// TIA Portal V21 export
DATA_BLOCK "Percorso"   // DB9
{ S7_Optimized_Access := 'TRUE' }
// stored: MemoryReserve 100
   VAR RETAIN
      Stazione { S7_SetPoint := 'True'} : Array[0.."K_NumStazione"] of "Std_Stazione";
   END_VAR
   VAR
      Hmi : Struct
         Visibilità : Struct
            PompaAcidificazioneVascaEvaporati : Struct
               VascaEvaporati : Bool := FALSE;
            END_STRUCT;
            Acidificazione1 : Struct
               Serpentino : Bool := FALSE;
               VascaPolpa1 : Bool := FALSE;
               VascaPolpa2 : Bool := FALSE;
            END_STRUCT;
            Acidificazione2 : Struct
               Serpentino : Bool := FALSE;
               VascaPolpa1 : Bool := FALSE;
               VascaPolpa2 : Bool := FALSE;
            END_STRUCT;
            Acidificazione3 : Struct
               Serpentino : Bool := FALSE;
               VascaPolpa1 : Bool := FALSE;
               VascaPolpa2 : Bool := FALSE;
               VascaMix : Bool := FALSE;
            END_STRUCT;
            Acidificazione4 : Struct
               Serpentino : Bool := FALSE;
               VascaPolpa1 : Bool := FALSE;
               VascaPolpa2 : Bool := FALSE;
            END_STRUCT;
            BermaProntoFresco : Struct
               CatelliLogicon : Bool := FALSE;
               CFT10t : Bool := FALSE;
               CatelliOhmico : Bool := FALSE;
               Goglio : Bool := FALSE;
            END_STRUCT;
            BermaPomodoro : Struct
               CatelliLogicon : Bool := FALSE;
               CFT10t : Bool := FALSE;
               CatelliOhmico : Bool := FALSE;
               Goglio : Bool := FALSE;
            END_STRUCT;
            Cernita1 : Struct
               IFT6 : Bool := FALSE;
               TrituratoD1 : Bool := FALSE;
            END_STRUCT;
            CFT_MVRAEstrazione1 : Struct
               VascaDecanter : Bool := FALSE;
               Vasca30Quintali : Bool := FALSE;
               VascaEvaporati : Bool := FALSE;
               CFT10t : Bool := FALSE;
               CatelliConcentrato : Bool := FALSE;
               CatelliOhmico : Bool := FALSE;
               BermaPomodoro : Bool := FALSE;
               BermaProntoFresco : Bool := FALSE;
               Ghizzoni : Bool := FALSE;
               PastorizzatoreGoglio2 : Bool := FALSE;
            END_STRUCT;
            CFT_MVRAEstrazione2 : Struct
               VascaDecanter : Bool := FALSE;
               Vasca30Quintali : Bool := FALSE;
               VascaEvaporati : Bool := FALSE;
               VascaSemiconcentrato : Bool := FALSE;
               CFT10t : Bool := FALSE;
               CatelliLogicon : Bool := FALSE;
               CatelliConcentrato : Bool := FALSE;
               CatelliOhmico : Bool := FALSE;
               Goglio : Bool := FALSE;
               BermaPomodoro : Bool := FALSE;
               BermaProntoFresco : Bool := FALSE;
               Ghizzoni : Bool := FALSE;
               PastorizzatoreGoglio2 : Bool := FALSE;
            END_STRUCT;
            CFT_MVRBEstrazione1 : Struct
               VascaDecanter : Bool := FALSE;
               Vasca30Quintali : Bool := FALSE;
               VascaPolpa1 : Bool := FALSE;
               VascaSemiconcentrato : Bool := FALSE;
               CFT10t : Bool := FALSE;
               CatelliLogicon : Bool := FALSE;
               CatelliOhmico : Bool := FALSE;
               Goglio : Bool := FALSE;
               BermaPomodoro : Bool := FALSE;
               BermaProntoFresco : Bool := FALSE;
               Ghizzoni : Bool := FALSE;
               PastorizzatoreGoglio2 : Bool := FALSE;
            END_STRUCT;
            CFT_MVRBFinitore1 : Struct
               VascaDecanter : Bool := FALSE;
               Vasca30Quintali : Bool := FALSE;
               VascaPolpa1 : Bool := FALSE;
               VascaSemiconcentrato : Bool := FALSE;
               CFT10t : Bool := FALSE;
               CatelliLogicon : Bool := FALSE;
               CatelliConcentrato : Bool := FALSE;
               CatelliOhmico : Bool := FALSE;
               Goglio : Bool := FALSE;
               BermaPomodoro : Bool := FALSE;
               BermaProntoFresco : Bool := FALSE;
               Ghizzoni : Bool := FALSE;
               PastorizzatoreGoglio2 : Bool := FALSE;
            END_STRUCT;
            CFT_MVRBFinitore2 : Struct
               VascaEvaporati : Bool := FALSE;
               CatelliConcentrato : Bool := FALSE;
               FBR200Kg : Bool := FALSE;
            END_STRUCT;
            CocleaIFT1_2 : Struct
               IFT1 : Bool := FALSE;
               IFT2 : Bool := FALSE;
            END_STRUCT;
            D1 : Struct
               PompaAlimentazioneHB1 : Bool := FALSE;
               PompaAlimentazioneHB2 : Bool := FALSE;
               PompaAlimentazioneHB1_HB2 : Bool := FALSE;
            END_STRUCT;
            D2 : Struct
               PompaAlimentazioneHB1 : Bool := FALSE;
               PompaAlimentazioneHB2 : Bool := FALSE;
               PompaAlimentazioneHB1_HB2 : Bool := FALSE;
            END_STRUCT;
            VascaDecanter1 : Struct
               VascaCrema : Bool := FALSE;
            END_STRUCT;
            VascaDecanter2 : Struct
               VascaCrema : Bool := FALSE;
            END_STRUCT;
            VascaDecanter3 : Struct
               VascaCrema : Bool := FALSE;
            END_STRUCT;
            Ghizzoni : Struct
               CFT10t : Bool := FALSE;
               CatelliLogicon : Bool := FALSE;
               CatelliOhmico : Bool := FALSE;
               Goglio : Bool := FALSE;
            END_STRUCT;
            IFT3 : Struct
               Lince1 : Bool := FALSE;
               Lince2 : Bool := FALSE;
               Lince3 : Bool := FALSE;
            END_STRUCT;
            IFT5 : Struct
               Lince1 : Bool := FALSE;
               Lince3 : Bool := FALSE;
            END_STRUCT;
            IFT6 : Struct
               Lince1 : Bool := FALSE;
               Lince2 : Bool := FALSE;
               Lince3 : Bool := FALSE;
            END_STRUCT;
            Lince1 : Struct
               Serpentino : Bool := FALSE;
               VascaPolpa1 : Bool := FALSE;
               VascaPolpa2 : Bool := FALSE;
            END_STRUCT;
            Lince2 : Struct
               Serpentino : Bool := FALSE;
               VascaPolpa1 : Bool := FALSE;
               VascaPolpa2 : Bool := FALSE;
            END_STRUCT;
            Lince3 : Struct
               Serpentino : Bool := FALSE;
               VascaPolpa1 : Bool := FALSE;
               VascaPolpa2 : Bool := FALSE;
               VascaMIx : Bool := FALSE;
            END_STRUCT;
            Lince4 : Struct
               Serpentino : Bool := FALSE;
               VascaPolpa1 : Bool := FALSE;
               VascaPolpa2 : Bool := FALSE;
            END_STRUCT;
            PICO1 : Struct
               CFT10t : Bool := FALSE;
               CatelliLogicon : Bool := FALSE;
               CatelliOhmico : Bool := FALSE;
               Goglio : Bool := FALSE;
               BermaPomodoro : Bool := FALSE;
               BermaProntoFresco : Bool := FALSE;
               Ghizzoni : Bool := FALSE;
               FBR200Kg : Bool := FALSE;
               PastorizzatoreGoglio2 : Bool := FALSE;
            END_STRUCT;
            PICO2 : Struct
               CFT10t : Bool := FALSE;
               CatelliLogicon : Bool := FALSE;
               CatelliConcentrato : Bool := FALSE;
               CatelliOhmico : Bool := FALSE;
               Goglio : Bool := FALSE;
               BermaPomodoro : Bool := FALSE;
               BermaProntoFresco : Bool := FALSE;
               Ghizzoni : Bool := FALSE;
               FBR200Kg : Bool := FALSE;
               PastorizzatoreGoglio2 : Bool := FALSE;
            END_STRUCT;
            PompaAlimentazioneDecanter : Struct
               VascaDecanter : Bool := FALSE;
            END_STRUCT;
            PompaAlimentazioneHB1 : Struct
               HB1 : Bool := FALSE;
               HB2 : Bool := FALSE;
            END_STRUCT;
            PompaAlimentazioneHB2 : Struct
               HB1 : Bool := FALSE;
               HB2 : Bool := FALSE;
               HB3 : Bool := FALSE;
            END_STRUCT;
            PompaAlimentazioneHB1_HB2 : Struct
               HB1 : Bool := FALSE;
               HB2 : Bool := FALSE;
            END_STRUCT;
            PompaAlimentazioneHB3 : Struct
               HB3 : Bool := FALSE;
            END_STRUCT;
            PompaInvio1 : Struct
               VascaMix : Bool := FALSE;
               CatelliConcentrato : Bool := FALSE;
               CatelliOhmico : Bool := FALSE;
               BermaPomodoro : Bool := FALSE;
               Ghizzoni : Bool := FALSE;
            END_STRUCT;
            PompaInvio2 : Struct
               CFT10t : Bool := FALSE;
               CatelliLogicon : Bool := FALSE;
               CatelliOhmico : Bool := FALSE;
               PastorizzatoreGoglio2 : Bool := FALSE;
               Ghizzoni : Bool := FALSE;
            END_STRUCT;
            PompaInvio3 : Struct
               FMCPolpa : Bool := FALSE;
               BermaPomodoro : Bool := FALSE;
            END_STRUCT;
            PompaInvio4 : Struct
               FMCPolpa : Bool := FALSE;
            END_STRUCT;
            PompaInvio5 : Struct
               CFT10t : Bool := FALSE;
               CatelliLogicon : Bool := FALSE;
               CatelliOhmico : Bool := FALSE;
               BermaPomodoro : Bool := FALSE;
               BermaProntoFresco : Bool := FALSE;
               Ghizzoni : Bool := FALSE;
               Goglio : Bool := FALSE;
            END_STRUCT;
            PompaInvio6 : Struct
               BermaProntoFresco : Bool := FALSE;
               Ghizzoni : Bool := FALSE;
               Goglio : Bool := FALSE;
               FBR200Kg : Bool := FALSE;
               PastorizzatoreGoglio2 : Bool := FALSE;
            END_STRUCT;
            PompaInvio7 : Struct
               CatelliLogicon : Bool := FALSE;
               CatelliOhmico : Bool := FALSE;
               Goglio : Bool := FALSE;
               BermaProntoFresco : Bool := FALSE;
               Ghizzoni : Bool := FALSE;
               FBR200Kg : Bool := FALSE;
               PastorizzatoreGoglio2 : Bool := FALSE;
            END_STRUCT;
            PompaNastroIFT1_2 : Struct
               D1 : Bool := FALSE;
               D2 : Bool := FALSE;
            END_STRUCT;
            PompaRecuperoIFT1 : Struct
               SgrondatoreP54 : Bool := FALSE;
               SgrondatoreP55 : Bool := FALSE;
            END_STRUCT;
            PompaRecuperoIFT2 : Struct
               SgrondatoreP54 : Bool := FALSE;
               SgrondatoreP55 : Bool := FALSE;
            END_STRUCT;
            PompaRecuperoPizza : Struct
               VascaDecanter : Bool := FALSE;
            END_STRUCT;
            Salsina1 : Struct
               Serpentino : Bool := FALSE;
               VascaPolpa1 : Bool := FALSE;
               VascaPolpa2 : Bool := FALSE;
            END_STRUCT;
            Salsina2 : Struct
               Serpentino : Bool := FALSE;
               VascaPolpa1 : Bool := FALSE;
               VascaPolpa2 : Bool := FALSE;
            END_STRUCT;
            Salsina3 : Struct
               Serpentino : Bool := FALSE;
               VascaPolpa1 : Bool := FALSE;
               VascaPolpa2 : Bool := FALSE;
               VascaMIx : Bool := FALSE;
            END_STRUCT;
            Salsina4 : Struct
               Serpentino : Bool := FALSE;
               VascaPolpa1 : Bool := FALSE;
               VascaPolpa2 : Bool := FALSE;
            END_STRUCT;
            Scrambler : Struct
               Lince1 : Bool := FALSE;
               Lince2 : Bool := FALSE;
               Lince3 : Bool := FALSE;
            END_STRUCT;
            Separapelli1Sx : Struct
               IFT3 : Bool := FALSE;
               IFT4 : Bool := FALSE;
               IFT5 : Bool := FALSE;
               Scrambler : Bool := FALSE;
            END_STRUCT;
            Separapelli2Dx : Struct
               IFT3 : Bool := FALSE;
               IFT4 : Bool := FALSE;
               IFT5 : Bool := FALSE;
               Scrambler : Bool := FALSE;
            END_STRUCT;
            Serpentino : Struct
               PompaInvio1 : Bool := FALSE;
               PompaInvio2 : Bool := FALSE;
               PompaInvio3 : Bool := FALSE;
               PompaInvio4 : Bool := FALSE;
               PompaInvio5 : Bool := FALSE;
            END_STRUCT;
            SgrondatoreP54 : Struct
               Lince1 : Bool := FALSE;
               Lince2 : Bool := FALSE;
               Lince3 : Bool := FALSE;
            END_STRUCT;
            SgrondatoreP55 : Struct
               Lince2 : Bool := FALSE;
               Lince3 : Bool := FALSE;
            END_STRUCT;
            "T150_1/2EffettoP05" : Struct
               VascaDecanter : Bool := FALSE;
               VascaEvaporati : Bool := FALSE;
               VascaPolpa1 : Bool := FALSE;
               Ghizzoni : Bool := FALSE;
               VascaSemiconcentrato : Bool := FALSE;
            END_STRUCT;
            "T150_1/2EffettoP07" : Struct
               VascaDecanter : Bool := FALSE;
               VascaEvaporati : Bool := FALSE;
               VascaPolpa1 : Bool := FALSE;
               CatelliOhmico : Bool := FALSE;
               Ghizzoni : Bool := FALSE;
               VascaSemiconcentrato : Bool := FALSE;
               BermaPomodoro : Bool := FALSE;
               BermaProntoFresco : Bool := FALSE;
            END_STRUCT;
            T150_3EffettofinitoreP02 : Struct
               VascaEvaporati : Bool := FALSE;
               VascaPolpa1 : Bool := FALSE;
               CatelliConcentrato : Bool := FALSE;
               CatelliOhmico : Bool := FALSE;
               VascaSemiconcentrato : Bool := FALSE;
               BermaPomodoro : Bool := FALSE;
               VascaDecanter : Bool := FALSE;
            END_STRUCT;
            TorchioSgrondatoreP54 : Struct
               Lince3 : Bool := FALSE;
            END_STRUCT;
            TorchioScrambler : Struct
               Lince1 : Bool := FALSE;
            END_STRUCT;
            TrituratoD1 : Struct
               D1 : Bool := FALSE;
            END_STRUCT;
            TrituratoD2 : Struct
               D2 : Bool := FALSE;
            END_STRUCT;
            TrituratoBrovatrice : Struct
               D1 : Bool := FALSE;
               D2 : Bool := FALSE;
            END_STRUCT;
            Vasca30Quintali : Struct
               Serpentino : Bool := FALSE;
            END_STRUCT;
            VascaDecanter : Struct
               VascaEvaporati : Bool := FALSE;
               Vasca30Quintali : Bool := FALSE;
               VascaPolpa1 : Bool := FALSE;
               Decanter1 : Bool := FALSE;
               Decanter2 : Bool := FALSE;
               Decanter3 : Bool := FALSE;
            END_STRUCT;
            VascaEvaporatiP134 : Struct
               CatelliOhmico : Bool := FALSE;
            END_STRUCT;
            VascaEvaporatiP135 : Struct
               CatelliConcentrato : Bool := FALSE;
            END_STRUCT;
            VascaMix : Struct
               PICO1 : Bool := FALSE;
               PICO2 : Bool := FALSE;
            END_STRUCT;
            VascaPolpa1 : Struct
               PompaInvio1 : Bool := FALSE;
               PompaInvio2 : Bool := FALSE;
               PompaInvio3 : Bool := FALSE;
               PompaInvio4 : Bool := FALSE;
               PompaInvio5 : Bool := FALSE;
               PompaInvio6 : Bool := FALSE;
               PompaInvio7 : Bool := FALSE;
            END_STRUCT;
            VascaPolpa2 : Struct
               PompaInvio1 : Bool := FALSE;
               PompaInvio2 : Bool := FALSE;
               PompaInvio3 : Bool := FALSE;
               PompaInvio4 : Bool := FALSE;
               PompaInvio5 : Bool := FALSE;
               PompaInvio6 : Bool := FALSE;
               PompaInvio7 : Bool := FALSE;
            END_STRUCT;
            PompaCrema1 : Struct
               CatelliConcentrato : Bool := FALSE;
               CatelliOhmico : Bool := FALSE;
               BermaPomodoro : Bool := FALSE;
               VascaMix : Bool := FALSE;
            END_STRUCT;
            PompaCrema2 : Struct
               CatelliLogicon : Bool := FALSE;
               CatelliOhmico : Bool := FALSE;
               CFT10t : Bool := FALSE;
            END_STRUCT;
            PompaCrema3 : Struct
               BermaPomodoro : Bool := FALSE;
               FMCPolpa : Bool := FALSE;
            END_STRUCT;
            PompaCrema4 : Struct
               FMCPolpa : Bool := FALSE;
            END_STRUCT;
            PompaCrema5 : Struct
               CFT10t : Bool := FALSE;
               CatelliLogicon : Bool := FALSE;
               CatelliOhmico : Bool := FALSE;
               Goglio : Bool := FALSE;
               BermaPomodoro : Bool := FALSE;
               BermaProntoFresco : Bool := FALSE;
               Ghizzoni : Bool := FALSE;
            END_STRUCT;
            IFT4 : Struct
               Lince2 : Bool := FALSE;
            END_STRUCT;
            PompaConcentrato1 : Struct
               VascaMix : Bool := FALSE;
            END_STRUCT;
         END_STRUCT;
         Comandi : Struct
            K_StazioneAttuale : Int := 0;
            RicercaSorgentiDest : Bool := FALSE;
            SceltaSorgDest_PopupAperto : Bool := FALSE;
            ElencoSorgentiPossibili : Array[0..15] of Int;
            ElencoDestinazioniPossibili : Array[0..15] of Int;
            SceltaTraSorgentiPossibili : Array[0..15] of Bool;
            SceltaTraDestinazioniPossibili : Array[0..15] of Bool;
            CaricaInLavoro : Bool := FALSE;
            ResettaTuttoOffline : Bool := FALSE;
            RipristinaOnline : Bool := FALSE;
            CompilaVerificaConflitti : Bool := FALSE;
         END_STRUCT;
      END_STRUCT;
   END_VAR
BEGIN
   // Stazione[0] : Non usare
   Stazione[0..1].IN.CodiceProdotto := 0;
   Stazione[0..1].IN.Portata := 0.0;
   Stazione[0..1].Prm.Partner.TipoAssociazione := 16#00;
   Stazione[0..1].Prm.CadutaChiamata.DaAnalogicaPer.SogliaMaxi := 16#00;
   Stazione[0..1].Prm.CadutaChiamata.DaAnalogicaPer.SogliaIntMax := 16#00;
   Stazione[0..1].Prm.CadutaChiamata.DaAnalogicaPer.SogliaIntMin := 16#00;
   Stazione[0..1].Prm.CadutaChiamata.DaAnalogicaPer.SogliaMini := 16#00;
   Stazione[0..1].Prm.BypassDestinazione := FALSE;
   Stazione[0..1].Prm.BypassSorgente := FALSE;
   Stazione[0..1].Hmi.Abilita := FALSE;
   Stazione[0..1].Hmi.ByPassConsensoMacchina := FALSE;
   Stazione[0..1].Hmi.Diagnostica."00-Analogica" := FALSE;
   Stazione[0..1].Hmi.Diagnostica."01-Paratia" := FALSE;
   Stazione[0..1].Hmi.Diagnostica."02-Motore" := FALSE;
   Stazione[0..1].Hmi.Diagnostica."03-Pompa" := FALSE;
   Stazione[0..1].Hmi.Diagnostica."04-NessunaStazioneInChiamata" := FALSE;
   Stazione[0..1].Hmi.Diagnostica."05-StopChiamataDaPLC" := FALSE;
   Stazione[0..1].Hmi.Diagnostica."06-SelettoreHMIStop" := FALSE;
   Stazione[0..1].Hmi.Diagnostica."07-MancanzaConsensoMacchina" := FALSE;
   Stazione[0..1].Hmi.Diagnostica."08-StazionePartnerNonChiama" := FALSE;
   Stazione[0..1].Hmi.Diagnostica."09-" := FALSE;
   Stazione[0..1].Allarmi.Stato.ConflittoMultiDest := FALSE;
   Stazione[0..1].Allarmi.EnWarnHmi.ConflittoMultiDest := FALSE;
   Stazione[0..1].Allarmi.WordHMI := 16#0000;
   Stazione[0].Destinazione[0].IN.Possibile := FALSE;   // Percorso selezionabile da HMI
   Stazione[0].Destinazione[1].IN.Possibile := FALSE;
   Stazione[1].Destinazione[0..1].IN.Possibile := FALSE;
   Stazione[0].Destinazione[0].IN.Selezionato := FALSE;   // Percorso selezionato e NON caricato online
   Stazione[0].Destinazione[1].IN.Selezionato := FALSE;
   Stazione[1].Destinazione[0..1].IN.Selezionato := FALSE;
   Stazione[0].Destinazione[0].IN.Attivo := FALSE;   // Percorso selezionato e caricato online
   Stazione[0].Destinazione[1].IN.Attivo := FALSE;
   Stazione[1].Destinazione[0..1].IN.Attivo := FALSE;
   Stazione[0].Destinazione[0..1].Prm.BypassChiamata := FALSE;
   Stazione[1].Destinazione[0..1].Prm.BypassChiamata := FALSE;
   Stazione[0..1].Dati.DestAttivaPresente := FALSE;
   Stazione[0..1].Dati.SorgAttivaPresente := FALSE;
   Stazione[0..1].Dati.AlmenoUnaSorgenteProgettata := FALSE;
   Stazione[0..1].Dati.AlmenoUnaDestinazioneProgettata := FALSE;
   Stazione[0..1].OUT.Chiamata := FALSE;
   Stazione[0..1].Rif_Inc.K_Analogica := 0;
   Stazione[0..1].Rif_Inc.K_Paratia := 0;
   Stazione[0..1].Rif_Inc.K_Motore := 0;
   Stazione[0..1].Rif_Inc.K_Pompa := 0;
   Stazione[0..1].Rif_Inc.K_Stazione := 0;
   Hmi.Comandi.ElencoSorgentiPossibili[0..15] := 0;
   Hmi.Comandi.ElencoDestinazioniPossibili[0..15] := 0;
   Hmi.Comandi.SceltaTraSorgentiPossibili[0..15] := FALSE;
   Hmi.Comandi.SceltaTraDestinazioniPossibili[0..15] := FALSE;
END_DATA_BLOCK
